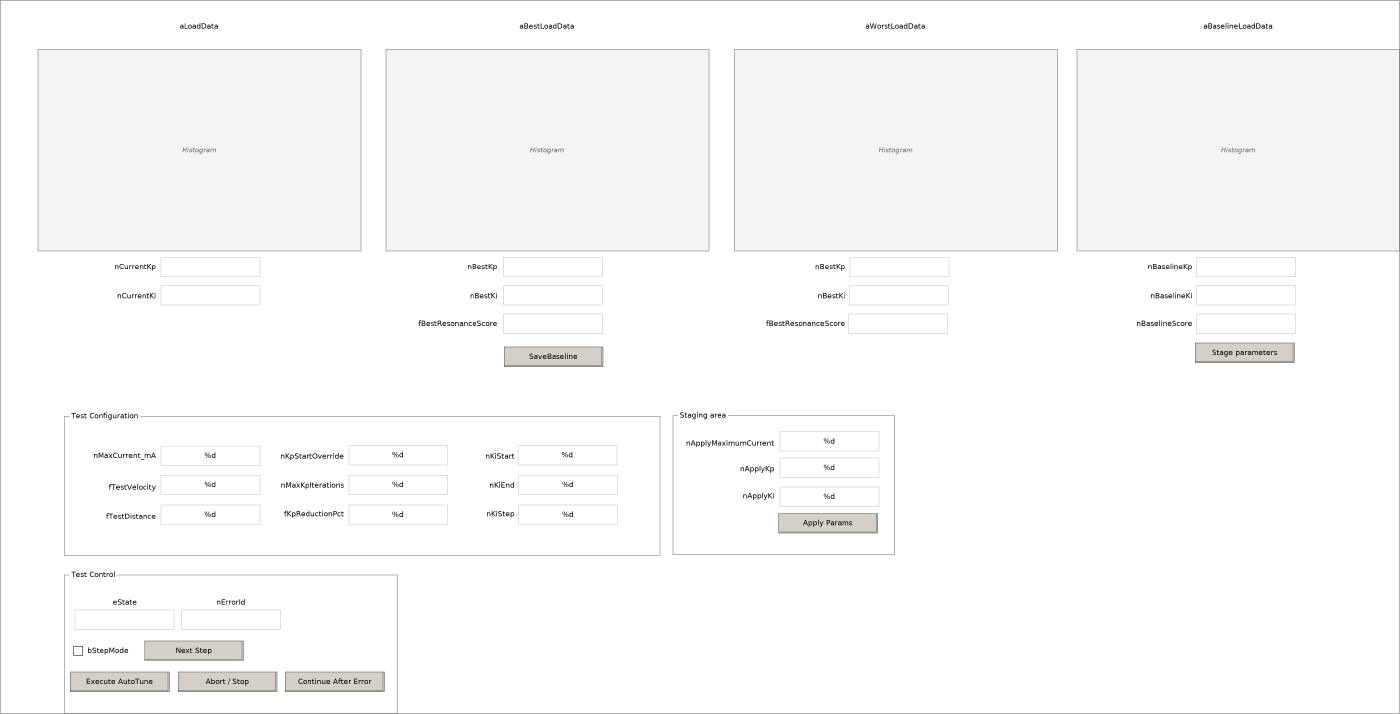
VISUALIZATION Visu_Tune_EL7047  // 2117x1081
VAR_IN_OUT
	fbTuner: FB_EL7047_Tuner;
END_VAR
    GroupBox (97,622 901x219), "Test Configuration"
    Button (106,1017 150x30), "Execute AutoTune", pressed state: fbTuner.bExecuteAutoTune
    Button (269,1017 150x30), "Abort / Stop", pressed state: fbTuner.bAbortTuning
    Button (431,1017 150x30), "Continue After Error", pressed state: fbTuner.bContinueAfterError
    Button (762,525 150x30), "SaveBaseline", pressed state: fbTuner.bSaveBaseline
    Button (1807,519 150x30), "Stage parameters", pressed state: fbTuner.bApplyParams
    Textfield (113,923 150x30), text variable: fbTuner.eState
    Textfield (274,923 150x30), text variable: fbTuner.nErrorId
    Textfield (243,389 150x30), text variable: fbTuner.nCurrentKp
    Textfield (243,432 150x30), text variable: fbTuner.nCurrentKi
    Textfield (761,389 150x30), text variable: fbTuner.nBestKp
    Textfield (761,432 150x30), text variable: fbTuner.nBestKi
    Textfield (761,475 150x30), text variable: fbTuner.fBestResonanceScore
    Textfield (1809,389 150x30), text variable: fbTuner.nBaselineKp
    Textfield (1809,432 150x30), text variable: fbTuner.nBaselineKi
    Textfield (1809,475 150x30), text variable: fbTuner.fBaselineScore
    Histogram (57,74 489x306), scale format: %.1f, scale -3000..3000
        p1518820177: fbTuner.aLoadData
        p102497268: fbTuner.aLoadData
        p788070771: ARRAY [1..5000] OF INT
    Histogram (1110,74 489x306), scale format: %.1f, scale -3000..3000
        p1518820177: fbTuner.aWorstLoadData
        p102497268: fbTuner.aWorstLoadData
        p788070771: ARRAY [1..5000] OF INT
    Histogram (1628,74 489x306), scale format: %.1f, scale -3000..3000
        p1518820177: fbTuner.aBaselineLoadData
        p102497268: fbTuner.aBaselineLoadData
        p788070771: ARRAY [1..5000] OF INT
    Label (114,897 150x30), "eState"
    Label (274,897 150x30), "nErrorId"
    Label (143,389 96x30), "nCurrentKp"
    Label (125,433 114x30), "nCurrentKi"
    Label (605,389 150x30), "nBestKp"
    Label (605,433 150x30), "nBestKi"
    Label (605,475 150x30), "fBestResonanceScore"
    Label (1656,389 150x30), "nBaselineKp"
    Label (1656,433 150x30), "nBaselineKi"
    Label (1656,475 150x30), "nBaselineScore"
    Label (226,25 150x30), "aLoadData"
    Label (752,25 150x30), "aBestLoadData"
    Label (1279,25 150x30), "aWorstLoadData"
    Label (1797,25 150x30), "aBaselineLoadData"
    Histogram (583,74 489x306), scale format: %.1f, scale -3000..3000
        p1518820177: fbTuner.aLoadData
        p102497268: fbTuner.aLoadData
        p788070771: ARRAY [1..5000] OF INT
    Textfield (1285,389 150x30), text variable: fbTuner.nBestKp
    Textfield (1284,432 150x30), text variable: fbTuner.nBestKi
    Textfield (1283,475 150x30), text variable: fbTuner.fBestResonanceScore
    Label (1131,389 150x30), "nBestKp"
    Label (1131,433 150x30), "nBestKi"
    Label (1131,475 150x30), "fBestResonanceScore"
    Textfield (527,674 150x30), "%d", text variable: fbTuner.nKpStartOverride
        OnMouseClick: write the text variable via Default
    Textfield (783,674 150x30), "%d", text variable: fbTuner.nKiStart
        OnMouseClick: write the text variable via Default
    Textfield (784,719 150x30), "%d", text variable: fbTuner.nKiEnd
        OnMouseClick: write the text variable via Default
    Textfield (784,764 150x30), "%d", text variable: fbTuner.nKiStep
        OnMouseClick: write the text variable via Default
    Textfield (527,719 150x30), "%d", text variable: fbTuner.nMaxKpIterations
        OnMouseClick: write the text variable via Default
    Textfield (527,764 150x30), "%d", text variable: fbTuner.fKpReductionPct
        OnMouseClick: write the text variable via Default
    Textfield (243,719 150x30), "%d", text variable: fbTuner.fTestVelocity
        OnMouseClick: write the text variable via Default
    Textfield (243,764 150x30), "%d", text variable: fbTuner.fTestDistance
        OnMouseClick: write the text variable via Default
    Label (143,675 96x30), "nMaxCurrent_mA"
    Textfield (243,675 150x30), "%d", text variable: fbTuner.nMaxCurrent_mA
        OnMouseClick: write the text variable via Default
    Label (427,676 96x30), "nKpStartOverride"
    Label (427,720 96x30), "nMaxKpIterations"
    Label (427,763 96x30), "fKpReductionPct"
    Label (729,676 52x30), "nKiStart"
    Label (728,720 53x30), "nKiEnd"
    Label (725,763 56x30), "nKiStep"
    Label (143,723 96x30), "fTestVelocity"
    Label (143,767 96x30), "fTestDistance"
    Textfield (1179,693 150x30), "%d", text variable: fbTuner.nApplyKp
        OnMouseClick: write the text variable via Default
    Textfield (1179,737 150x30), "%d", text variable: fbTuner.nApplyKi
        OnMouseClick: write the text variable via Default
    Label (1122,695 52x30), "nApplyKp"
    Label (1122,736 52x30), "nApplyKi"
    Textfield (1179,653 150x30), "%d", text variable: fbTuner.nApplyM
        OnMouseClick: write the text variable via Default
    Label (1033,656 141x30), "nApplyMaximumCurrent"
    Button (1177,777 150x30), "Apply Params", pressed state: fbTuner.bApplyParams
    GroupBox (1017,621 336x219), "Staging area"
    Checkbox (109,970 150x30), "bStepMode", variable: fbTuner.bStepMode
    Button (218,970 150x30), "Next Step", pressed state: fbTuner.bNextStep
    GroupBox (97,862 504x219), "Test Control"
END_VISUALIZATION

(* stored: Version 1.1.0.1
   Visu Visu_Tune_EL7047: Id {c64305f7-7a98-0942-2292-11f0626db71c} *)
